// TwinCAT 3 PLC project UrsaPQ_PLC
// ProgramVersion: 3.1.4022.4
// libraries:
//   Tc2_MC2, * (Beckhoff Automation GmbH)
//   Tc2_Standard, * (Beckhoff Automation GmbH)
//   Tc2_System, * (Beckhoff Automation GmbH)
//   Tc3_Module, * (Beckhoff Automation GmbH)
// project tree:
//   GVLs/ GVL.TcGVL, POU.TcPOU (not stored)
//   / PlcTask.TcTTO
//   POUs/ ConvertPressure_Pirani.TcPOU, MAIN.TcPOU, PressureChamber_MNG.TcPOU, manageAxis.TcPOU, ConvertPressure_Penning.TcPOU, PARAM.TcGVL
// real-time tasks:
//   TASK PlcTask: cycle T#5ms, priority 20, ADS port 350
// motion (NC):
//   TASK NC-Task SAF: cycle T#2ms, priority 4, ADS port 501
//   TASK NC-Task SVB: cycle T#10ms, priority 8, ADS port 511
//   AXIS FrameX (id 1)
//     General: UnitName=s
//     Dynamic: AccelerationMaximum=5000, Acceleration=7.99999, Deceleration=7.99999
//     Velo: RefSearch=0.5, RefSync=0.5, Maximum=0.5
//     OtherSettings: AllowMotionCmdToSlave=true
//     encoder EncType=4
//       EncPara: MaxCount=#x0000ffff
//         Inc: RefSoftSyncMask=#x0000ffff
//     drive DrvType=24
//       Analog: VeloReferenz=12.8, ScaleFactorActTorque=0.1
//       TimeComp: TaskDelayCycles=1
//     controller CtrType=1
//       CtrPara: PriorControlFactor=1
//         PID: PosKp=5
//         Observer: BandWidth=20
//   AXIS FrameY (id 2)
//     Dynamic: AccelerationMaximum=5000, Acceleration=8, Deceleration=8
//     Velo: Maximum=2
//     OtherSettings: AllowMotionCmdToSlave=true
//     encoder EncType=4
//       EncPara: MaxCount=#x0000ffff
//         Inc: RefSoftSyncMask=#x0000ffff
//     drive DrvType=24
//       Analog: VeloReferenz=12.8, ScaleFactorActTorque=0.1
//       TimeComp: TaskDelayCycles=1
//     controller CtrType=1
//       CtrPara: PriorControlFactor=1
//         PID: PosKp=5
//         Observer: BandWidth=20
//   AXIS SampleX (id 3)
//     Dynamic: AccelerationMaximum=5000, Acceleration=8, Deceleration=8
//     Velo: SlowManual=1, FastManual=2, Maximum=2
//     OtherSettings: AllowMotionCmdToSlave=true, PulseDistancePos=1, PulseDistanceNeg=1
//     encoder EncType=4
//       EncPara: MaxCount=#x0000ffff
//         Inc: RefSoftSyncMask=#x0000ffff
//     drive DrvType=24
//       Analog: VeloReferenz=12.8, ScaleFactorActTorque=0.1
//       TimeComp: TaskDelayCycles=1
//     controller CtrType=1
//       CtrPara: PriorControlFactor=1
//         PosDiffControl: Range=10
//         PID: PosKp=2
//         Observer: BandWidth=20
//   AXIS SampleY (id 4)
//     Dynamic: AccelerationMaximum=5000, Acceleration=8, Deceleration=8
//     Velo: SlowManual=1, FastManual=2, Maximum=2
//     OtherSettings: AllowMotionCmdToSlave=true, PulseDistancePos=1, PulseDistanceNeg=1
//     encoder EncType=4
//       EncPara: MaxCount=#x0000ffff
//         Inc: RefSoftSyncMask=#x0000ffff
//     drive DrvType=24
//       Analog: VeloReferenz=12.8, ScaleFactorActTorque=0.1
//       TimeComp: TaskDelayCycles=1
//     controller CtrType=1
//       CtrPara: PriorControlFactor=1
//         Observer: BandWidth=20
//   AXIS SampleZ (id 5)
//     Dynamic: Acceleration=8, Deceleration=8
//     Velo: RefSearch=60, RefSync=60, SlowManual=1, FastManual=4, Maximum=10
//     OtherSettings: AllowMotionCmdToSlave=true, DataPersistence=true, PulseDistancePos=1, PulseDistanceNeg=1
//     encoder EncType=4
//       EncPara: MaxCount=#x0000ffff
//         Inc: RefMode=1, RefSoftSyncMask=#x0000ffff
//     drive DrvType=24
//       Analog: VeloReferenz=12.8, ScaleFactorActTorque=0.1
//       TimeComp: TaskDelayCycles=1
//     controller CtrType=1
//       CtrPara: PriorControlFactor=1
//         PID: PosKp=20
//         Observer: BandWidth=20
//   AXIS Magnet Y (id 6)
//     Dynamic: Acceleration=8, Deceleration=8
//     Velo: SlowManual=1, FastManual=2, Maximum=2
//     OtherSettings: AllowMotionCmdToSlave=true, PulseDistancePos=1, PulseDistanceNeg=1
//     encoder EncType=4
//       EncPara: MaxCount=#x0000ffff
//         Inc: RefSoftSyncMask=#x0000ffff
//     drive DrvType=24
//       Analog: VeloReferenz=12.8, ScaleFactorActTorque=0.1
//       TimeComp: TaskDelayCycles=1
//     controller CtrType=1
//       CtrPara: PriorControlFactor=1
//         PID: PosKp=20
//         Observer: BandWidth=20
// I/O:
//   DEVICE Device 3 (EtherCAT), AmsNetId 172.18.237.166.4.1
//     Term 1 (EK1100) [EK1100 EtherCAT Coupler (2A E-Bus)]
//       Term 2 Frame X (EL7047) [EL7047 1Ch. Stepper motor output stage (50V, 5A)]
//       Term 3 Frame Y  (EL7047) [EL7047 1Ch. Stepper motor output stage (50V, 5A)]
//       Term 4 Sample X (EL7047) [EL7047 1Ch. Stepper motor output stage (50V, 5A)]
//       Term 5 Sample Y (EL7047) [EL7047 1Ch. Stepper motor output stage (50V, 5A)]
//       Term 6 Sample Z (EL7047) [EL7047 1Ch. Stepper motor output stage (50V, 5A)]
//       Term 7 Magnet Y (EL7047) [EL7047 1Ch. Stepper motor output stage (50V, 5A)]
//       Term 8 (EL9576) [EL9576 Brake chopper terminal]
//       LVPS + M1 Valve [EL2602-0010 2Ch. Relay Output + ZCD, NO (230V AC / 30V DC)]
//       Valves M2 + TOF [EL2602-0010 2Ch. Relay Output + ZCD, NO (230V AC / 30V DC)]
//       Lamp1 [EL2602-0010 2Ch. Relay Output + ZCD, NO (230V AC / 30V DC)]
//       Term 46 (EL9011) [EL9011 End Terminal]
//     Term 27 (EK1100) [EK1100 EtherCAT Coupler (2A E-Bus)]
//       Oven Supply [EL2596 1-channel LED strobe control terminal 24V/3A]
//       Coil Supply [EL2596 1-channel LED strobe control terminal 24V/3A]
//       Pirani Gauges [EL3164 4Ch. Ana. Input 0-10V]
//       Penning Gauges + FlowValve [EL3164 4Ch. Ana. Input 0-10V]
//       TurboTOF_enable + penning enable [EL2004 4Ch. Dig. Output 24V, 0.5A]
//       Term 32 (EL1008) [EL1008 8Ch. Dig. Input 24V, 3ms]
//       TurboTOF Input [EL1819 16Ch. Dig. Input 24V, 10µs]
//       Term 37 (EL3318) [EL3318 8Ch. Ana Input Thermocouple (TC)]
//       Flow Valve Control [EL4002 2Ch. Ana. Output 0-10V, 12bit]
//       Profibus [EL6731 PROFIBUS DP Master]
//       Term 40 (EL6022) [EL6022 Interface 2Ch. (RS422/485)]
//       Term 49 (EL9011) [EL9011 End Terminal]
//     Term 38 (EK1100) [EK1100 EtherCAT Coupler (2A E-Bus)]
//       HVPS PowerSupply [EL4012 2Ch. Ana. Output 0-20mA, 12bit]
//       FlashInterlock [EL2004 4Ch. Dig. Output 24V, 0.5A]
//       Term 48 (EL9011) [EL9011 End Terminal]
//   DEVICE Device 2 (EL6731), AmsNetId 192.168.0.1.3.1
//     Box 10 (GSD Box) (Anybus-CC Profibus-DPV1) // Vendor: HMS Industrial Networks Revision: 1.02
// variable links:
//   NC-Task SAF/Axes/FrameX <-> Device 3 (EtherCAT)/Term 1 (EK1100)/Term 2 Frame X (EL7047)
//     Drive/Inputs/In/nState1 @bit 3 <-> STM Status/Status/Error
//     Drive/Inputs/In/nState1 @bit 7 <-> STM Status/Status/Motor stall
//     Drive/Inputs/In/nState1 @bit 5 <-> STM Status/Status/Moving negative
//     Drive/Inputs/In/nState1 @bit 4 <-> STM Status/Status/Moving positive
//     Drive/Inputs/In/nState1 @bit 1 <-> STM Status/Status/Ready
//     Drive/Inputs/In/nState1 <-> STM Status/Status/Ready to enable
//     Drive/Inputs/In/nState1 @bit 6 <-> STM Status/Status/Torque reduced
//     Drive/Inputs/In/nState1 @bit 2 <-> STM Status/Status/Warning
//     Drive/Inputs/In/nState2 @bit 5 <-> STM Status/Status/Sync error
//     Drive/Inputs/In/nState2 @bit 7 <-> STM Status/Status/TxPDO Toggle
//     Drive/Inputs/In/nState4 @bit 1 <-> WcState/InputToggle
//     Drive/Inputs/In/nState4 <-> WcState/WcState
//     Drive/Outputs/Out/nCtrl1 <-> STM Control/Control/Enable
//     Drive/Outputs/Out/nCtrl1 @bit 2 <-> STM Control/Control/Reduce torque
//     Drive/Outputs/Out/nCtrl1 @bit 1 <-> STM Control/Control/Reset
//     Drive/Outputs/Out/nCtrl2 @bit 3 <-> STM Control/Control/Digital output 1
//     Drive/Outputs/Out/nDataOut2[0] <-> STM Velocity/Velocity
//     Enc/Inputs/In/nDataIn1[0] <-> ENC Status compact/Counter value
//     Enc/Inputs/In/nDataIn2[0] <-> ENC Status compact/Latch value
//     Enc/Inputs/In/nState1 @bit 4 <-> ENC Status compact/Status/Counter overflow
//     Enc/Inputs/In/nState1 @bit 3 <-> ENC Status compact/Status/Counter underflow
//     Enc/Inputs/In/nState1 @bit 7 <-> ENC Status compact/Status/Extrapolation stall
//     Enc/Inputs/In/nState1 <-> ENC Status compact/Status/Latch C valid
//     Enc/Inputs/In/nState1 @bit 1 <-> ENC Status compact/Status/Latch extern valid
//     Enc/Inputs/In/nState1 @bit 2 <-> ENC Status compact/Status/Set counter done
//     Enc/Inputs/In/nState2 @bit 4 <-> ENC Status compact/Status/Status of extern latch
//     Enc/Inputs/In/nState2 <-> ENC Status compact/Status/Status of input A
//     Enc/Inputs/In/nState2 @bit 1 <-> ENC Status compact/Status/Status of input B
//     Enc/Inputs/In/nState2 @bit 2 <-> ENC Status compact/Status/Status of input C
//     Enc/Inputs/In/nState2 @bit 5 <-> ENC Status compact/Status/Sync error
//     Enc/Inputs/In/nState2 @bit 7 <-> ENC Status compact/Status/TxPDO Toggle
//     Enc/Inputs/In/nState4 @bit 1 <-> WcState/InputToggle
//     Enc/Inputs/In/nState4 <-> WcState/WcState
//     Enc/Outputs/Out/nCtrl1 <-> ENC Control compact/Control/Enable latch C
//     Enc/Outputs/Out/nCtrl1 @bit 3 <-> ENC Control compact/Control/Enable latch extern on negative edge
//     Enc/Outputs/Out/nCtrl1 @bit 1 <-> ENC Control compact/Control/Enable latch extern on positive edge
//     Enc/Outputs/Out/nCtrl1 @bit 2 <-> ENC Control compact/Control/Set counter
//     Enc/Outputs/Out/nDataOut1[0] <-> ENC Control compact/Set counter value
//   NC-Task SAF/Axes/FrameY <-> Device 3 (EtherCAT)/Term 1 (EK1100)/Term 3 Frame Y  (EL7047)
//     Drive/Inputs/In/nState1 @bit 3 <-> STM Status/Status/Error
//     Drive/Inputs/In/nState1 @bit 7 <-> STM Status/Status/Motor stall
//     Drive/Inputs/In/nState1 @bit 5 <-> STM Status/Status/Moving negative
//     Drive/Inputs/In/nState1 @bit 4 <-> STM Status/Status/Moving positive
//     Drive/Inputs/In/nState1 @bit 1 <-> STM Status/Status/Ready
//     Drive/Inputs/In/nState1 <-> STM Status/Status/Ready to enable
//     Drive/Inputs/In/nState1 @bit 6 <-> STM Status/Status/Torque reduced
//     Drive/Inputs/In/nState1 @bit 2 <-> STM Status/Status/Warning
//     Drive/Inputs/In/nState2 @bit 5 <-> STM Status/Status/Sync error
//     Drive/Inputs/In/nState2 @bit 7 <-> STM Status/Status/TxPDO Toggle
//     Drive/Inputs/In/nState4 @bit 1 <-> WcState/InputToggle
//     Drive/Inputs/In/nState4 <-> WcState/WcState
//     Drive/Outputs/Out/nCtrl1 <-> STM Control/Control/Enable
//     Drive/Outputs/Out/nCtrl1 @bit 2 <-> STM Control/Control/Reduce torque
//     Drive/Outputs/Out/nCtrl1 @bit 1 <-> STM Control/Control/Reset
//     Drive/Outputs/Out/nCtrl2 @bit 3 <-> STM Control/Control/Digital output 1
//     Drive/Outputs/Out/nDataOut2[0] <-> STM Velocity/Velocity
//     Enc/Inputs/In/nDataIn1[0] <-> ENC Status compact/Counter value
//     Enc/Inputs/In/nDataIn2[0] <-> ENC Status compact/Latch value
//     Enc/Inputs/In/nState1 @bit 4 <-> ENC Status compact/Status/Counter overflow
//     Enc/Inputs/In/nState1 @bit 3 <-> ENC Status compact/Status/Counter underflow
//     Enc/Inputs/In/nState1 @bit 7 <-> ENC Status compact/Status/Extrapolation stall
//     Enc/Inputs/In/nState1 <-> ENC Status compact/Status/Latch C valid
//     Enc/Inputs/In/nState1 @bit 1 <-> ENC Status compact/Status/Latch extern valid
//     Enc/Inputs/In/nState1 @bit 2 <-> ENC Status compact/Status/Set counter done
//     Enc/Inputs/In/nState2 @bit 4 <-> ENC Status compact/Status/Status of extern latch
//     Enc/Inputs/In/nState2 <-> ENC Status compact/Status/Status of input A
//     Enc/Inputs/In/nState2 @bit 1 <-> ENC Status compact/Status/Status of input B
//     Enc/Inputs/In/nState2 @bit 2 <-> ENC Status compact/Status/Status of input C
//     Enc/Inputs/In/nState2 @bit 5 <-> ENC Status compact/Status/Sync error
//     Enc/Inputs/In/nState2 @bit 7 <-> ENC Status compact/Status/TxPDO Toggle
//     Enc/Inputs/In/nState4 @bit 1 <-> WcState/InputToggle
//     Enc/Inputs/In/nState4 <-> WcState/WcState
//     Enc/Outputs/Out/nCtrl1 <-> ENC Control compact/Control/Enable latch C
//     Enc/Outputs/Out/nCtrl1 @bit 3 <-> ENC Control compact/Control/Enable latch extern on negative edge
//     Enc/Outputs/Out/nCtrl1 @bit 1 <-> ENC Control compact/Control/Enable latch extern on positive edge
//     Enc/Outputs/Out/nCtrl1 @bit 2 <-> ENC Control compact/Control/Set counter
//     Enc/Outputs/Out/nDataOut1[0] <-> ENC Control compact/Set counter value
//   NC-Task SAF/Axes/Magnet Y <-> Device 3 (EtherCAT)/Term 1 (EK1100)/Term 7 Magnet Y (EL7047)
//     Drive/Inputs/In/nState1 @bit 3 <-> STM Status/Status/Error
//     Drive/Inputs/In/nState1 @bit 7 <-> STM Status/Status/Motor stall
//     Drive/Inputs/In/nState1 @bit 5 <-> STM Status/Status/Moving negative
//     Drive/Inputs/In/nState1 @bit 4 <-> STM Status/Status/Moving positive
//     Drive/Inputs/In/nState1 @bit 1 <-> STM Status/Status/Ready
//     Drive/Inputs/In/nState1 <-> STM Status/Status/Ready to enable
//     Drive/Inputs/In/nState1 @bit 6 <-> STM Status/Status/Torque reduced
//     Drive/Inputs/In/nState1 @bit 2 <-> STM Status/Status/Warning
//     Drive/Inputs/In/nState2 @bit 5 <-> STM Status/Status/Sync error
//     Drive/Inputs/In/nState2 @bit 7 <-> STM Status/Status/TxPDO Toggle
//     Drive/Inputs/In/nState4 @bit 1 <-> WcState/InputToggle
//     Drive/Inputs/In/nState4 <-> WcState/WcState
//     Drive/Outputs/Out/nCtrl1 <-> STM Control/Control/Enable
//     Drive/Outputs/Out/nCtrl1 @bit 2 <-> STM Control/Control/Reduce torque
//     Drive/Outputs/Out/nCtrl1 @bit 1 <-> STM Control/Control/Reset
//     Drive/Outputs/Out/nCtrl2 @bit 3 <-> STM Control/Control/Digital output 1
//     Drive/Outputs/Out/nDataOut2[0] <-> STM Velocity/Velocity
//     Enc/Inputs/In/nDataIn1[0] <-> ENC Status compact/Counter value
//     Enc/Inputs/In/nDataIn2[0] <-> ENC Status compact/Latch value
//     Enc/Inputs/In/nState1 @bit 4 <-> ENC Status compact/Status/Counter overflow
//     Enc/Inputs/In/nState1 @bit 3 <-> ENC Status compact/Status/Counter underflow
//     Enc/Inputs/In/nState1 @bit 7 <-> ENC Status compact/Status/Extrapolation stall
//     Enc/Inputs/In/nState1 <-> ENC Status compact/Status/Latch C valid
//     Enc/Inputs/In/nState1 @bit 1 <-> ENC Status compact/Status/Latch extern valid
//     Enc/Inputs/In/nState1 @bit 2 <-> ENC Status compact/Status/Set counter done
//     Enc/Inputs/In/nState2 @bit 4 <-> ENC Status compact/Status/Status of extern latch
//     Enc/Inputs/In/nState2 <-> ENC Status compact/Status/Status of input A
//     Enc/Inputs/In/nState2 @bit 1 <-> ENC Status compact/Status/Status of input B
//     Enc/Inputs/In/nState2 @bit 2 <-> ENC Status compact/Status/Status of input C
//     Enc/Inputs/In/nState2 @bit 5 <-> ENC Status compact/Status/Sync error
//     Enc/Inputs/In/nState2 @bit 7 <-> ENC Status compact/Status/TxPDO Toggle
//     Enc/Inputs/In/nState4 @bit 1 <-> WcState/InputToggle
//     Enc/Inputs/In/nState4 <-> WcState/WcState
//     Enc/Outputs/Out/nCtrl1 <-> ENC Control compact/Control/Enable latch C
//     Enc/Outputs/Out/nCtrl1 @bit 3 <-> ENC Control compact/Control/Enable latch extern on negative edge
//     Enc/Outputs/Out/nCtrl1 @bit 1 <-> ENC Control compact/Control/Enable latch extern on positive edge
//     Enc/Outputs/Out/nCtrl1 @bit 2 <-> ENC Control compact/Control/Set counter
//     Enc/Outputs/Out/nDataOut1[0] <-> ENC Control compact/Set counter value
//   NC-Task SAF/Axes/SampleX <-> Device 3 (EtherCAT)/Term 1 (EK1100)/Term 4 Sample X (EL7047)
//     Drive/Inputs/In/nState1 @bit 3 <-> STM Status/Status/Error
//     Drive/Inputs/In/nState1 @bit 7 <-> STM Status/Status/Motor stall
//     Drive/Inputs/In/nState1 @bit 5 <-> STM Status/Status/Moving negative
//     Drive/Inputs/In/nState1 @bit 4 <-> STM Status/Status/Moving positive
//     Drive/Inputs/In/nState1 @bit 1 <-> STM Status/Status/Ready
//     Drive/Inputs/In/nState1 <-> STM Status/Status/Ready to enable
//     Drive/Inputs/In/nState1 @bit 6 <-> STM Status/Status/Torque reduced
//     Drive/Inputs/In/nState1 @bit 2 <-> STM Status/Status/Warning
//     Drive/Inputs/In/nState2 @bit 5 <-> STM Status/Status/Sync error
//     Drive/Inputs/In/nState2 @bit 7 <-> STM Status/Status/TxPDO Toggle
//     Drive/Inputs/In/nState4 @bit 1 <-> WcState/InputToggle
//     Drive/Inputs/In/nState4 <-> WcState/WcState
//     Drive/Outputs/Out/nCtrl1 <-> STM Control/Control/Enable
//     Drive/Outputs/Out/nCtrl1 @bit 2 <-> STM Control/Control/Reduce torque
//     Drive/Outputs/Out/nCtrl1 @bit 1 <-> STM Control/Control/Reset
//     Drive/Outputs/Out/nCtrl2 @bit 3 <-> STM Control/Control/Digital output 1
//     Drive/Outputs/Out/nDataOut2[0] <-> STM Velocity/Velocity
//     Enc/Inputs/In/nDataIn1[0] <-> ENC Status compact/Counter value
//     Enc/Inputs/In/nDataIn2[0] <-> ENC Status compact/Latch value
//     Enc/Inputs/In/nState1 @bit 4 <-> ENC Status compact/Status/Counter overflow
//     Enc/Inputs/In/nState1 @bit 3 <-> ENC Status compact/Status/Counter underflow
//     Enc/Inputs/In/nState1 @bit 7 <-> ENC Status compact/Status/Extrapolation stall
//     Enc/Inputs/In/nState1 <-> ENC Status compact/Status/Latch C valid
//     Enc/Inputs/In/nState1 @bit 1 <-> ENC Status compact/Status/Latch extern valid
//     Enc/Inputs/In/nState1 @bit 2 <-> ENC Status compact/Status/Set counter done
//     Enc/Inputs/In/nState2 @bit 4 <-> ENC Status compact/Status/Status of extern latch
//     Enc/Inputs/In/nState2 <-> ENC Status compact/Status/Status of input A
//     Enc/Inputs/In/nState2 @bit 1 <-> ENC Status compact/Status/Status of input B
//     Enc/Inputs/In/nState2 @bit 2 <-> ENC Status compact/Status/Status of input C
//     Enc/Inputs/In/nState2 @bit 5 <-> ENC Status compact/Status/Sync error
//     Enc/Inputs/In/nState2 @bit 7 <-> ENC Status compact/Status/TxPDO Toggle
//     Enc/Inputs/In/nState4 @bit 1 <-> WcState/InputToggle
//     Enc/Inputs/In/nState4 <-> WcState/WcState
//     Enc/Outputs/Out/nCtrl1 <-> ENC Control compact/Control/Enable latch C
//     Enc/Outputs/Out/nCtrl1 @bit 3 <-> ENC Control compact/Control/Enable latch extern on negative edge
//     Enc/Outputs/Out/nCtrl1 @bit 1 <-> ENC Control compact/Control/Enable latch extern on positive edge
//     Enc/Outputs/Out/nCtrl1 @bit 2 <-> ENC Control compact/Control/Set counter
//     Enc/Outputs/Out/nDataOut1[0] <-> ENC Control compact/Set counter value
//   NC-Task SAF/Axes/SampleY <-> Device 3 (EtherCAT)/Term 1 (EK1100)/Term 5 Sample Y (EL7047)
//     Drive/Inputs/In/nState1 @bit 3 <-> STM Status/Status/Error
//     Drive/Inputs/In/nState1 @bit 7 <-> STM Status/Status/Motor stall
//     Drive/Inputs/In/nState1 @bit 5 <-> STM Status/Status/Moving negative
//     Drive/Inputs/In/nState1 @bit 4 <-> STM Status/Status/Moving positive
//     Drive/Inputs/In/nState1 @bit 1 <-> STM Status/Status/Ready
//     Drive/Inputs/In/nState1 <-> STM Status/Status/Ready to enable
//     Drive/Inputs/In/nState1 @bit 6 <-> STM Status/Status/Torque reduced
//     Drive/Inputs/In/nState1 @bit 2 <-> STM Status/Status/Warning
//     Drive/Inputs/In/nState2 @bit 5 <-> STM Status/Status/Sync error
//     Drive/Inputs/In/nState2 @bit 7 <-> STM Status/Status/TxPDO Toggle
//     Drive/Inputs/In/nState4 @bit 1 <-> WcState/InputToggle
//     Drive/Inputs/In/nState4 <-> WcState/WcState
//     Drive/Outputs/Out/nCtrl1 <-> STM Control/Control/Enable
//     Drive/Outputs/Out/nCtrl1 @bit 2 <-> STM Control/Control/Reduce torque
//     Drive/Outputs/Out/nCtrl1 @bit 1 <-> STM Control/Control/Reset
//     Drive/Outputs/Out/nCtrl2 @bit 3 <-> STM Control/Control/Digital output 1
//     Drive/Outputs/Out/nDataOut2[0] <-> STM Velocity/Velocity
//     Enc/Inputs/In/nDataIn1[0] <-> ENC Status compact/Counter value
//     Enc/Inputs/In/nDataIn2[0] <-> ENC Status compact/Latch value
//     Enc/Inputs/In/nState1 @bit 4 <-> ENC Status compact/Status/Counter overflow
//     Enc/Inputs/In/nState1 @bit 3 <-> ENC Status compact/Status/Counter underflow
//     Enc/Inputs/In/nState1 @bit 7 <-> ENC Status compact/Status/Extrapolation stall
//     Enc/Inputs/In/nState1 <-> ENC Status compact/Status/Latch C valid
//     Enc/Inputs/In/nState1 @bit 1 <-> ENC Status compact/Status/Latch extern valid
//     Enc/Inputs/In/nState1 @bit 2 <-> ENC Status compact/Status/Set counter done
//     Enc/Inputs/In/nState2 @bit 4 <-> ENC Status compact/Status/Status of extern latch
//     Enc/Inputs/In/nState2 <-> ENC Status compact/Status/Status of input A
//     Enc/Inputs/In/nState2 @bit 1 <-> ENC Status compact/Status/Status of input B
//     Enc/Inputs/In/nState2 @bit 2 <-> ENC Status compact/Status/Status of input C
//     Enc/Inputs/In/nState2 @bit 5 <-> ENC Status compact/Status/Sync error
//     Enc/Inputs/In/nState2 @bit 7 <-> ENC Status compact/Status/TxPDO Toggle
//     Enc/Inputs/In/nState4 @bit 1 <-> WcState/InputToggle
//     Enc/Inputs/In/nState4 <-> WcState/WcState
//     Enc/Outputs/Out/nCtrl1 <-> ENC Control compact/Control/Enable latch C
//     Enc/Outputs/Out/nCtrl1 @bit 3 <-> ENC Control compact/Control/Enable latch extern on negative edge
//     Enc/Outputs/Out/nCtrl1 @bit 1 <-> ENC Control compact/Control/Enable latch extern on positive edge
//     Enc/Outputs/Out/nCtrl1 @bit 2 <-> ENC Control compact/Control/Set counter
//     Enc/Outputs/Out/nDataOut1[0] <-> ENC Control compact/Set counter value
//   NC-Task SAF/Axes/SampleZ <-> Device 3 (EtherCAT)/Term 1 (EK1100)/Term 6 Sample Z (EL7047)
//     Drive/Inputs/In/nState1 @bit 3 <-> STM Status/Error
//     Drive/Inputs/In/nState1 @bit 7 <-> STM Status/Motor stall
//     Drive/Inputs/In/nState1 @bit 5 <-> STM Status/Moving negative
//     Drive/Inputs/In/nState1 @bit 4 <-> STM Status/Moving positive
//     Drive/Inputs/In/nState1 @bit 1 <-> STM Status/Ready
//     Drive/Inputs/In/nState1 <-> STM Status/Ready to enable
//     Drive/Inputs/In/nState1 @bit 6 <-> STM Status/Torque reduced
//     Drive/Inputs/In/nState1 @bit 2 <-> STM Status/Warning
//     Drive/Inputs/In/nState2 @bit 5 <-> STM Status/Sync error
//     Drive/Inputs/In/nState2 @bit 7 <-> STM Status/TxPDO Toggle
//     Drive/Inputs/In/nState4 @bit 1 <-> WcState/InputToggle
//     Drive/Inputs/In/nState4 <-> WcState/WcState
//     Drive/Outputs/Out/nCtrl1 <-> STM Control/Enable
//     Drive/Outputs/Out/nCtrl1 @bit 2 <-> STM Control/Reduce torque
//     Drive/Outputs/Out/nCtrl1 @bit 1 <-> STM Control/Reset
//     Drive/Outputs/Out/nCtrl2 @bit 3 <-> STM Control/Digital output 1
//     Drive/Outputs/Out/nDataOut2[0] <-> STM Velocity/Velocity
//     Enc/Inputs/In/nDataIn1[0] <-> ENC Status compact/Counter value
//     Enc/Inputs/In/nDataIn2[0] <-> ENC Status compact/Latch value
//     Enc/Inputs/In/nState1 @bit 4 <-> ENC Status compact/Counter overflow
//     Enc/Inputs/In/nState1 @bit 3 <-> ENC Status compact/Counter underflow
//     Enc/Inputs/In/nState1 @bit 7 <-> ENC Status compact/Extrapolation stall
//     Enc/Inputs/In/nState1 <-> ENC Status compact/Latch C valid
//     Enc/Inputs/In/nState1 @bit 1 <-> ENC Status compact/Latch extern valid
//     Enc/Inputs/In/nState1 @bit 2 <-> ENC Status compact/Set counter done
//     Enc/Inputs/In/nState2 @bit 4 <-> ENC Status compact/Status of extern latch
//     Enc/Inputs/In/nState2 <-> ENC Status compact/Status of input A
//     Enc/Inputs/In/nState2 @bit 1 <-> ENC Status compact/Status of input B
//     Enc/Inputs/In/nState2 @bit 2 <-> ENC Status compact/Status of input C
//     Enc/Inputs/In/nState2 @bit 5 <-> ENC Status compact/Sync error
//     Enc/Inputs/In/nState2 @bit 7 <-> ENC Status compact/TxPDO Toggle
//     Enc/Inputs/In/nState4 @bit 1 <-> WcState/InputToggle
//     Enc/Inputs/In/nState4 <-> WcState/WcState
//     Enc/Outputs/Out/nCtrl1 <-> ENC Control compact/Enable latch C
//     Enc/Outputs/Out/nCtrl1 @bit 3 <-> ENC Control compact/Enable latch extern on negative edge
//     Enc/Outputs/Out/nCtrl1 @bit 1 <-> ENC Control compact/Enable latch extern on positive edge
//     Enc/Outputs/Out/nCtrl1 @bit 2 <-> ENC Control compact/Set counter
//     Enc/Outputs/Out/nDataOut1[0] <-> ENC Control compact/Set counter value
//   UrsaPQ_PLC/UrsaPQ_PLC Instance <-> Device 2 (EL6731)/Box 10 (GSD Box) (Anybus-CC Profibus-DPV1)
//     PlcTask Inputs/MAIN.TurboMain_ERR <-> Module 1 (PPO1)/Inputs/PPO1_0_1[0] @bit 11
//     PlcTask Inputs/MAIN.TurboMain_Freq <-> Module 1 (PPO1)/Inputs/PPO1_0_1[1]
//     PlcTask Inputs/MAIN.TurboMain_NO <-> Module 1 (PPO1)/Inputs/PPO1_0_1[0] @bit 2
//     PlcTask Inputs/MAIN.TurboMain_Overtemp <-> Module 1 (PPO1)/Inputs/PPO1_0_1[0] @bit 15
//     PlcTask Outputs/MAIN.TurboMain_Control <-> Module 1 (PPO1)/Outputs/PPO1_1_1[0] @bit 2
//     PlcTask Outputs/MAIN.TurboMain_enable <-> Module 1 (PPO1)/Outputs/PPO1_1_1[0] @bit 8
//   UrsaPQ_PLC/UrsaPQ_PLC Instance <-> Device 3 (EtherCAT)/Term 1 (EK1100)/LVPS + M1 Valve
//     PlcTask Outputs/MAIN.LVPS_ON <-> Channel 1/LVPS
//     PlcTask Outputs/MAIN.MPreVac_Valve <-> Channel 2/MainPrevacValve
//   UrsaPQ_PLC/UrsaPQ_PLC Instance <-> Device 3 (EtherCAT)/Term 1 (EK1100)/Lamp1
//     PlcTask Outputs/MAIN.Lamp1_Enable <-> Channel 1/Lamp1
//   UrsaPQ_PLC/UrsaPQ_PLC Instance <-> Device 3 (EtherCAT)/Term 1 (EK1100)/Term 2 Frame X (EL7047)
//     PlcTask Inputs/MAIN.FrameX_Bw_End <-> STM Status/Status/Digital input 2
//     PlcTask Inputs/MAIN.FrameX_Fw_End <-> STM Status/Status/Digital input 1
//   UrsaPQ_PLC/UrsaPQ_PLC Instance <-> Device 3 (EtherCAT)/Term 1 (EK1100)/Term 3 Frame Y  (EL7047)
//     PlcTask Inputs/MAIN.FrameY_Bw_End <-> STM Status/Status/Digital input 2
//     PlcTask Inputs/MAIN.FrameY_Fw_End <-> STM Status/Status/Digital input 1
//   UrsaPQ_PLC/UrsaPQ_PLC Instance <-> Device 3 (EtherCAT)/Term 1 (EK1100)/Term 4 Sample X (EL7047)
//     PlcTask Inputs/MAIN.SampleX_Bw_End <-> STM Status/Status/Digital input 1
//     PlcTask Inputs/MAIN.SampleX_Fw_End <-> STM Status/Status/Digital input 2
//   UrsaPQ_PLC/UrsaPQ_PLC Instance <-> Device 3 (EtherCAT)/Term 1 (EK1100)/Term 5 Sample Y (EL7047)
//     PlcTask Inputs/MAIN.SampleY_Bw_End <-> STM Status/Status/Digital input 1
//     PlcTask Inputs/MAIN.SampleY_Fw_End <-> STM Status/Status/Digital input 2
//   UrsaPQ_PLC/UrsaPQ_PLC Instance <-> Device 3 (EtherCAT)/Term 1 (EK1100)/Term 6 Sample Z (EL7047)
//     PlcTask Inputs/MAIN.SampleZ_Bw_End <-> STM Status/Digital input 2
//     PlcTask Inputs/MAIN.SampleZ_Fw_End <-> STM Status/Digital input 1
//   UrsaPQ_PLC/UrsaPQ_PLC Instance <-> Device 3 (EtherCAT)/Term 1 (EK1100)/Term 7 Magnet Y (EL7047)
//     PlcTask Inputs/MAIN.MagnetY_Bw_End <-> STM Status/Status/Digital input 2
//     PlcTask Inputs/MAIN.MagnetY_Fw_End <-> STM Status/Status/Digital input 1
//   UrsaPQ_PLC/UrsaPQ_PLC Instance <-> Device 3 (EtherCAT)/Term 1 (EK1100)/Valves M2 + TOF
//     PlcTask Outputs/MAIN.TOFPreVac_Valve <-> Channel 2/TOFPreVacValve
//   UrsaPQ_PLC/UrsaPQ_PLC Instance <-> Device 3 (EtherCAT)/Term 27 (EK1100)/Coil Supply
//     PlcTask Inputs/MAIN.Coil_Curr_In <-> DOX Synchron info data/Info data 2
//     PlcTask Inputs/MAIN.Coil_Err <-> DOX Status/Error
//     PlcTask Outputs/MAIN.Coil_Curr_Out <-> DOX Current/Output current
//     PlcTask Outputs/MAIN.Coil_Enable <-> DOX Control/Enable
//     PlcTask Outputs/MAIN.Coil_Output <-> DOX Control/Output
//     PlcTask Outputs/MAIN.Coil_Reset <-> DOX Control/Reset
//   UrsaPQ_PLC/UrsaPQ_PLC Instance <-> Device 3 (EtherCAT)/Term 27 (EK1100)/Flow Valve Control
//     PlcTask Outputs/MAIN.Flow_Valve_Set <-> AO Outputs Channel 1/Flow Valve Control
//   UrsaPQ_PLC/UrsaPQ_PLC Instance <-> Device 3 (EtherCAT)/Term 27 (EK1100)/Penning Gauges + FlowValve
//     PlcTask Inputs/MAIN.Chamber_Penning_Int <-> AI Standard Channel 1/Chamber Penning
//   UrsaPQ_PLC/UrsaPQ_PLC Instance <-> Device 3 (EtherCAT)/Term 27 (EK1100)/Pirani Gauges
//     PlcTask Inputs/MAIN.Chamber_Pirani_Int <-> AI Standard Channel 3/Chamber Pirani
//     PlcTask Inputs/MAIN.Flow_Valve <-> AI Standard Channel 4/Flow Valve
//     PlcTask Inputs/MAIN.GasLine_Pirani_Int <-> AI Standard Channel 2/Gas Delivery Line
//     PlcTask Inputs/MAIN.PrePump_Pressure_Int <-> AI Standard Channel 1/Prepump Pirani
//   UrsaPQ_PLC/UrsaPQ_PLC Instance <-> Device 3 (EtherCAT)/Term 27 (EK1100)/Term 37 (EL3318)
//     PlcTask Inputs/MAIN.Magnet_Temp <-> TC Channel 8/Magnet
//     PlcTask Inputs/MAIN.Sample_BodyTemp <-> TC Channel 3/Body
//     PlcTask Inputs/MAIN.Sample_CapTemp <-> TC Channel 2/Cap
//     PlcTask Inputs/MAIN.Sample_TipTemp <-> TC Channel 4/Tip2
//   UrsaPQ_PLC/UrsaPQ_PLC Instance <-> Device 3 (EtherCAT)/Term 27 (EK1100)/TurboTOF Input
//     PlcTask Inputs/MAIN.TurboTOF_ERR <-> Channel 10/TurboTOF_ERR
//     PlcTask Inputs/MAIN.TurboTOF_NO <-> Channel 2/TurboTOF_NO
//   UrsaPQ_PLC/UrsaPQ_PLC Instance <-> Device 3 (EtherCAT)/Term 27 (EK1100)/TurboTOF_enable + penning enable
//     PlcTask Outputs/MAIN.Penning_Enable <-> Channel 1/Penning Enable
//     PlcTask Outputs/MAIN.TurboTOF_enable <-> Channel 4/TurboTOF_enable
//   UrsaPQ_PLC/UrsaPQ_PLC Instance <-> Device 3 (EtherCAT)/Term 38 (EK1100)/FlashInterlock
//     PlcTask Outputs/MAIN.FlashInterlock <-> Channel 1/FlashInterlock
//   UrsaPQ_PLC/UrsaPQ_PLC Instance <-> Device 3 (EtherCAT)/Term 38 (EK1100)/HVPS PowerSupply
//     PlcTask Outputs/MAIN.HVPS_ON <-> AO Outputs Channel 1/HVPS Safety Loop
//   UrsaPQ_PLC/UrsaPQ_PLC Instance <-> NC-Task SAF/Axes/FrameX
//     PlcTask Inputs/MAIN.FrameX.NcToPlc <-> Outputs/ToPlc
//     PlcTask Outputs/MAIN.FrameX.PlcToNc <-> Inputs/FromPlc
//   UrsaPQ_PLC/UrsaPQ_PLC Instance <-> NC-Task SAF/Axes/FrameY
//     PlcTask Inputs/MAIN.FrameY.NcToPlc <-> Outputs/ToPlc
//     PlcTask Outputs/MAIN.FrameY.PlcToNc <-> Inputs/FromPlc
//   UrsaPQ_PLC/UrsaPQ_PLC Instance <-> NC-Task SAF/Axes/Magnet Y
//     PlcTask Inputs/MAIN.MagnetY.NcToPlc <-> Outputs/ToPlc
//     PlcTask Outputs/MAIN.MagnetY.PlcToNc <-> Inputs/FromPlc
//   UrsaPQ_PLC/UrsaPQ_PLC Instance <-> NC-Task SAF/Axes/SampleX
//     PlcTask Inputs/MAIN.SampleX.NcToPlc <-> Outputs/ToPlc
//     PlcTask Outputs/MAIN.SampleX.PlcToNc <-> Inputs/FromPlc
//   UrsaPQ_PLC/UrsaPQ_PLC Instance <-> NC-Task SAF/Axes/SampleY
//     PlcTask Inputs/MAIN.SampleY.NcToPlc <-> Outputs/ToPlc
//     PlcTask Outputs/MAIN.SampleY.PlcToNc <-> Inputs/FromPlc
//   UrsaPQ_PLC/UrsaPQ_PLC Instance <-> NC-Task SAF/Axes/SampleZ
//     PlcTask Inputs/MAIN.SampleZ.NcToPlc <-> Outputs/ToPlc
//     PlcTask Outputs/MAIN.SampleZ.PlcToNc <-> Inputs/FromPlc

CONFIGURATION UrsaPQ_PLC
    RESOURCE PLC ON TwinCAT3
        TASK PlcTask(INTERVAL := T#5ms, PRIORITY := 20);
        PROGRAM MAIN WITH PlcTask : MAIN;
    END_RESOURCE
END_CONFIGURATION

// ---- GVLs/GVL.TcGVL
{attribute 'qualified_only'}
VAR_GLOBAL
END_VAR

// ---- POUs/PARAM.TcGVL
{attribute 'qualified_only'}
VAR_GLOBAL CONSTANT
	PreVac_Ok_Threshold  : REAL := 2.5E0;   // mBar
	MainVac_Ok_Threshold : REAL := 2E-6;    // mBar
	TurboStart_Threshold : REAL := 2E0;     // mBar

	PenningMix_Start : REAL := 6E-3; //mBar (Enable penning and mixes the pirani with penning vals)
	PenningMix_End   : REAL := 6E-4; //mBar (Stops mixing and uses penning only)
        
	Sample_Movement_Speed: REAL := 2;
	Sample_Movement_Speed_Z: REAL := 5; 
	Frame_Movement_Speed : REAL := 0.2;
	
	Oven_MaxTemp : INT := 2500; // 200 deg C
	HVPS_SafetyLoop_Current : INT := 15000;
END_VAR

// ---- POUs/MAIN.TcPOU
PROGRAM MAIN
VAR		
	//**********************************************************INPUTS
	PrePump_Pressure_Int AT %I* : INT;
	Chamber_Penning_Int  AT %I* : INT;
	Chamber_Pirani_Int   AT %I* : INT;	
	GasLine_Pirani_Int   AT %I* : INT;
	Sample_BodyTemp      AT %I* : INT;					// Oven temperatures in 0.01 degC
	Sample_CapTemp       AT %I* : INT;
	Sample_TipTemp       AT %I* : INT;	
	Magnet_Temp          AT %I* : INT;
	
	Flow_Valve 			 AT %I* : INT;                  // Gas flow valve conductance 0-10 V
	
	TurboTOF_NO AT %I* : BOOL;	
	TurboTOF_ERR AT %I* : BOOL;
		
	// IMPORTANT! 
	// LEYBOLD AND BECKHOOF PLC USE DIFFERENT BYTE ORDER, be careful when linking to profibus
	// LEYBOLD:   0  1  2  3  4  5  6  7  8  9  10 11 12 13 14 15
	// BECKHOFF:  8  9  10 11 12 13 14 15 0  1  2  3  4  5  6  7 
	TurboMain_Overtemp AT %I* : BOOL;
	TurboMain_NO AT %I* : BOOL;
	TurboMain_ERR AT %I* : BOOL;
	TurboMain_Freq AT %I* : UINT;
	
	Coil_Err AT %I* : BOOL;
	Coil_Curr_In AT %I* : INT;
	
	
	//**************************************************************OUTPUTS
	Coil_Enable AT %Q* : BOOL;
	Coil_Output AT %Q* : BOOL;
	Coil_Reset AT %Q* : BOOL;
	Coil_Curr_Out AT %Q* : INT;

	Penning_Enable AT %Q* : BOOL;
	LVPS_ON AT %Q* : BOOL;
	MPreVac_Valve AT %Q*: BOOL;
	TOFPreVac_Valve AT %Q* : BOOL;

	TurboTOF_enable AT %Q* : BOOL;
	TurboMain_enable AT %Q*: BOOL;
	TurboMain_Control AT %Q* : BOOL;

	Flow_Valve_Set AT %Q* : INT;    // Flow valve setpoint
	
	FlashInterlock AT %Q* : BOOL;	
	HVPS_ON AT %Q* : INT;
	Lamp1_Enable AT %Q* : BOOL;
	
	//************************************ ADS inputs: CONTROL PARAMETERS (PLC reads values and acts accordignly, ADS clients should set these values)
	GasLine_Enable :    BOOL := FALSE;
	Pumps_Enable :      BOOL := FALSE;      // Start pumping sequence
	PreVac_Valve_Lock : BOOL := FALSE;		// Ovverides auto valves and close prevac valves
	
	Sample_Flow_Set : REAL := 0;
	
	SampleX_MotionEnable : BOOL := FALSE;     // Motion enables and setpoints input
	SampleY_MotionEnable : BOOL := FALSE;  	
	SampleZ_MotionEnable : BOOL := FALSE;  	
	SampleX_MotionStop    : BOOL := FALSE;
	SampleY_MotionStop    : BOOL := FALSE;
	SampleZ_MotionStop    : BOOL := FALSE;
	
	FrameX_MotionEnable  : BOOL := FALSE;
	FrameY_MotionEnable  : BOOL := FALSE;
	FrameX_MotionStop     : BOOL := FALSE;
	FrameY_MotionStop     : BOOL := FALSE;
	
	MagnetY_MotionEnable : BOOL := FALSE;
	MagnetY_MotionStop    : BOOL := FALSE;
	
	SampleX_SetPoint : REAL := 0;
	SampleY_SetPoint : REAL := 0;
	SampleZ_SetPoint : REAL := 0;
	FrameX_SetPoint  : REAL := 0;
	FrameY_SetPoint  : REAL := 0;
	MagnetY_SetPoint  : REAL := 0;
	
	//******************************************* ADS outputs: READ ONLY (PLC updates them at every cycle, ADS clients should just read)
	Chamber_Pressure : REAL;				// Main chamber pressure in mBars
	GasLine_Pressure : REAL;
	PreVac_Pressure  : REAL;                // PrePump line pressure
	PreVacValves_Open: BOOL;	            // Are valves open?

	Sample_Flow : REAL;
	
	TurboPump_ON: BOOL;
	TurboError: BOOL;	
	Turbo_NO:    BOOL;
	
	//Other vars
	PreVac_OK :  BOOL;						// Good prevacuum 
	MainVac_OK : BOOL;
	MainVac_TurboOK : BOOL;
	Oven_OverTEMP: BOOL;
	Pressure_Chamber_Manager: PressureChamber_MNG;
	
	//MOTION 
	manageAx_SampleX: manageAxis;
	manageAx_SampleY: manageAxis;
	manageAx_SampleZ: manageAxis;
	manageAx_FrameX: manageAxis;
	manageAx_FrameY: manageAxis;
	manageAx_MagnetY: manageAxis;	
		
	FrameX : AXIS_REF;
	FrameY : AXIS_REF;
	SampleZ : AXIS_REF;
	SampleX : AXIS_REF;
	SampleY : AXIS_REF;
	MagnetY : AXIS_REF;
	
	SampleX_Fw_End AT %I* : BOOL; // Limit switches
	SampleX_Bw_End AT %I* : BOOL;
	SampleY_Fw_End AT %I* : BOOL;
	SampleY_Bw_End AT %I* : BOOL; 
	SampleZ_Fw_End AT %I* : BOOL;
	SampleZ_Bw_End AT %I* : BOOL;  
	
	FrameX_Fw_End AT %I* : BOOL;
	FrameX_Bw_End AT %I* : BOOL; 
	FrameY_Fw_End AT %I* : BOOL;
	FrameY_Bw_End AT %I* : BOOL; 
	
	MagnetY_Fw_End AT %I* : BOOL;
	MagnetY_Bw_End AT %I* : BOOL;
END_VAR

//*** PROCESS INPUTS ***
//Get pressures in mbar (from ADC value)
Pressure_Chamber_Manager(penningInt := Chamber_Penning_Int, piraniInt := Chamber_Pirani_Int, penningOn => Penning_enable, pressureOut => Chamber_Pressure);
PreVac_Pressure := ConvertPressure_Pirani(PrePump_Pressure_Int);
GasLine_Pressure := ConvertPressure_Pirani(GasLine_Pirani_Int);

//*** MOTION ***
//Move axes
manageAx_SampleX(axis := SampleX, setPoint := SampleX_SetPoint, speed := PARAM.Sample_Movement_Speed, 
		 enable := SampleX_MotionEnable, stop:= SampleX_MotionStop, fwLimit := SampleX_Fw_End, bwLimit := SampleX_Bw_End);
		 
manageAx_SampleY(axis := SampleY, setPoint := SampleY_SetPoint, speed := PARAM.Sample_Movement_Speed, 
		 enable := SampleY_MotionEnable, stop:= SampleY_MotionStop, fwLimit := SampleY_Fw_End, bwLimit := SampleY_Bw_End);	 

manageAx_SampleZ(axis := SampleZ, setPoint := SampleZ_SetPoint, speed := PARAM.Sample_Movement_Speed_Z, 
		 enable := SampleZ_MotionEnable, stop:= SampleZ_MotionStop, fwLimit := SampleZ_Fw_End, bwLimit := SampleZ_Bw_End);
		 
manageAx_FrameX(axis := FrameX,  setPoint := FrameX_SetPoint,  speed := PARAM.Frame_Movement_Speed , 
		 enable := FrameX_MotionEnable, stop:= FrameX_MotionStop, fwLimit := FrameX_Fw_End,  bwLimit := FrameX_Bw_End);

manageAx_FrameY(axis := FrameY,  setPoint := FrameY_SetPoint,  speed := PARAM.Frame_Movement_Speed , 
		 enable := FrameY_MotionEnable, stop:= FrameY_MotionStop, fwLimit := FrameY_Fw_End,  bwLimit := FrameY_Bw_End);
		 
manageAx_MagnetY(axis := MagnetY, setPoint := MagnetY_SetPoint, speed := PARAM.Sample_Movement_Speed, 
		 enable := MagnetY_MotionEnable, stop:= MagnetY_MotionStop, fwLimit := MagnetY_Fw_End, bwLimit := MagnetY_Bw_End);
		 
		 
//*** SAFETY CHECKS ***
// Compute status variables
Oven_OverTEMP   := Sample_BodyTemp > PARAM.Oven_MaxTemp OR Sample_TipTemp > PARAM.Oven_MaxTemp OR Sample_CapTemp > PARAM.Oven_MaxTemp; // Prevent overtemp of oven
TurboError 		:= TurboTOF_ERR AND TurboMain_ERR;
Turbo_NO        := TurboTOF_NO AND TurboMain_NO; 
MainVac_OK      := Chamber_Pressure > 0 AND Chamber_Pressure < PARAM.MainVac_Ok_Threshold; // Negative pressure means sensor error or sensor disconnected
MainVac_TurboOK := Chamber_Pressure > 0 AND Chamber_Pressure < PARAM.TurboStart_Threshold;
PreVac_OK       := PreVac_Pressure  > 0 AND PreVac_Pressure  < PARAM.PreVac_Ok_Threshold;

Coil_Output := TRUE;
IF Coil_Reset THEN
	Coil_Reset := FALSE;
END_IF
IF Coil_Err THEN  // If coil error, disable the coil and reset
	Coil_Enable := FALSE;
	Coil_Reset := TRUE;
END_IF


// Decide actions based on status
PreVacValves_Open := NOT PreVac_Valve_Lock AND ( PreVac_OK OR NOT MainVac_TurboOK );
TurboPump_ON := PreVac_Ok AND Pumps_Enable AND MainVac_TurboOK AND NOT TurboError;
LVPS_ON := MainVac_TurboOK AND NOT Oven_OverTEMP;

// Sample Valve
Sample_Flow := INT_TO_REAL(Flow_Valve) / 32767; // convert int to float in range 0-1
Sample_Flow_Set := MAX( MIN( Sample_Flow_Set, 1), 0);
Flow_Valve_Set := REAL_TO_INT( Sample_Flow_Set * 32767) * BOOL_TO_INT(GasLine_Enable) * BOOL_TO_INT(MainVac_TurboOK);  // If vented, valve is closed

// Actuate outputs (when one action controls more than one output)
MPreVac_Valve   := PreVacValves_Open;
TOFPreVac_Valve := PreVacValves_Open;
TurboTOF_enable  := TurboPump_ON;
TurboMain_enable := TurboPump_ON;
TurboMain_control := TRUE; // Tell pump that control is through Profibus and ignore other signals

IF MainVac_OK AND Turbo_NO THEN
	FlashInterlock := TRUE;
	HVPS_ON := PARAM.HVPS_SafetyLoop_Current;
ELSE
	FlashInterlock := FALSE;
	HVPS_ON := 0;
END_IF

END_PROGRAM

// ---- POUs/PressureChamber_MNG.TcPOU
FUNCTION_BLOCK PressureChamber_MNG
VAR_INPUT
	penningInt : INT;
	piraniInt : INT;
END_VAR
VAR_OUTPUT
	penningON : BOOL;
	pressureOut: REAL;
END_VAR
VAR
	voltage : REAL;
	penningPressure: REAL;
	piraniPressure: REAL;
	mix: REAL;
END_VAR

piraniPressure := ConvertPressure_Pirani(piraniInt);

IF piraniPressure > PARAM.PenningMix_Start THEN
	pressureOut := piraniPressure;
	penningON := FALSE;
ELSE
	penningON := TRUE;
	penningPressure := ConvertPressure_Penning(penningInt);
	mix := ( piraniPressure - PARAM.PenningMix_End ) / (PARAM.PenningMix_Start - PARAM.PenningMix_End);
	IF mix < 0 THEN
		mix := 0;
	END_IF
	pressureOut := mix * piraniPressure + ( 1 - mix) * penningPressure;
END_IF

END_FUNCTION_BLOCK

// ---- POUs/ConvertPressure_Pirani.TcPOU
FUNCTION ConvertPressure_Pirani : REAL
VAR_INPUT
	pressureInt : INT;
END_VAR
VAR
	voltage: REAL;
END_VAR

voltage :=  pressureInt / 3276.8;

IF voltage < 0.5 THEN
	ConvertPressure_Pirani := 1000; //ERROR (SENSOR DISCONNECTED??)
ELSE
	ConvertPressure_Pirani := EXPT(10, ( voltage - 6.143 ) / 1.286 ); // Converts ADC integer to mbars (formula from thermovac manual)
END_IF

END_FUNCTION

// ---- POUs/ConvertPressure_Penning.TcPOU
FUNCTION ConvertPressure_Penning : REAL
VAR_INPUT
	penningInt: INT;
END_VAR
VAR
	voltage: LREAL;
END_VAR

//IF voltage < 1.5 OR NOT enabled THEN
//	ConvertPressure_Penning := -1; //ERROR (SENSOR DISCONNECTED??)
//ELSE
//	IF voltage > 9.6 THEN
//		voltage := 9.6;
//	END_IF
//	ConvertPressure_Penning := EXPT(10, ( voltage - 12.86 ) / 1.33 ); // voltage to mbars (formula from Leybold penningvac manual)
//END_IF

//Pfeiffer Penning routine
voltage :=  penningInt / 3276.8;

IF voltage < 2.0 THEN
	ConvertPressure_Penning := 1000; //ERROR (SENSOR DISCONNECTED??)
ELSE
	IF voltage > 8.6 THEN
		voltage := 8.6;
	END_IF
	ConvertPressure_Penning := EXPT(10, ( 1.25 * voltage - 12.75 )); // voltage to mbars (formula from Pfeiffer penningvac IKR 270 manual)
END_IF

END_FUNCTION

// ---- POUs/manageAxis.TcPOU
FUNCTION_BLOCK manageAxis
VAR_IN_OUT
	axis: AXIS_REF;
	enable: BOOL;
	stop : BOOL;
END_VAR
VAR_INPUT
	speed: REAL;
	fwLimit: BOOL;
	bwLimit: BOOL;
	setPoint : REAL;
END_VAR
VAR
	mcPower : MC_Power;
	mcAbs : MC_MoveAbsolute;
	mcHalt : MC_Halt;
	mcStop : MC_Stop;
	mcSetPos : MC_SetPosition;
END_VAR

// Takes an axis and a set point and gives the appropriate commands to the NC task to move the motor

// Enable / Disable motion based on enable state and limit switches status
mcPower( Axis:= axis, Enable:= TRUE,
	     Enable_Positive:= NOT fwLimit, Enable_Negative:= NOT bwLimit, Override:= 100);
		 
// Reset position if a end switch is set ('homing function')
//mcSetPos(Axis := axis, Execute := bwLimit, Position := 0);

// Move if new setpoint is requested		 
IF enable THEN     // If current set point is different from input value, trigger enable rising edge for MC_MoveAbsolute
	mcHalt (Axis:= axis, Execute := TRUE);  // Halts eventual motion command still in progress
	mcAbs(  Axis:= axis, Execute:= TRUE,    // Starts new motion
		    Position:= setPoint, Velocity:= speed);
	enable := FALSE;
ELSE										      // Bring enable down while waiting for next movement
	mcAbs(  Axis:= axis, Execute:= FALSE,
		    Position:= setPoint, Velocity:= speed);
END_IF			


mcStop (Axis:= axis, Execute := stop);  // Used to stop motion

END_FUNCTION_BLOCK
